// TIA Portal V18 export
// export: Created 2021-05-25T13:42:38.8465497Z, ExportSetting WithDefaults, WithReadOnly, DisplayName Totally Integrated Automation Portal, DisplayVersion V18, DisplayName TIA Portal Openness, DisplayVersion V18, DisplayName TIA Portal Version Control Interface, DisplayVersion V18, DisplayName Feature Cycle 1 TIA Portal, DisplayVersion V18, DisplayName STEP 7 Professional, DisplayVersion V18, DisplayName SIMATIC Energy Suite, DisplayVersion V18, DisplayName STEP 7 Safety, DisplayVersion V18, DisplayName WinCC Professional, DisplayVersion V18
ORGANIZATION_BLOCK "Main"   // OB1, LAD, ProgramCycle
TITLE = "Main Program Sweep (Cycle)"
{ S7_Optimized_Access := 'TRUE' }
VERSION : 0.1
// stored: AutoNumber true, CodeModifiedDate 2021-05-25T13:42:20.5536351Z, CompileDate 2021-05-25T13:42:38.4564505Z, ConstantName OB_Main, CreationDate 2021-05-25T13:31:11.728453Z, EventClass Program cycle, HandleErrorsWithinBlock false, InterfaceModifiedDate 2008-07-21T16:55:08.419547Z, IsConsistent true, IsIECCheckEnabled false, IsKnowHowProtected false, IsWriteProtected false, ModifiedDate 2021-05-25T13:42:20.5536351Z, ParameterModified 2008-07-21T16:55:08.419547Z, PLCSimAdvancedSupport false, PriorityNumber 1, ProcessImagePartNumber 65535, SetENOAutomatically false, StructureModified 2008-07-21T16:55:08.419547Z
   VAR_INPUT
      Initial_Call : Bool;   // Initial call of this OB
      Remanence : Bool;   // =True, if remanent data are available
   END_VAR
BEGIN
END_ORGANIZATION_BLOCK
